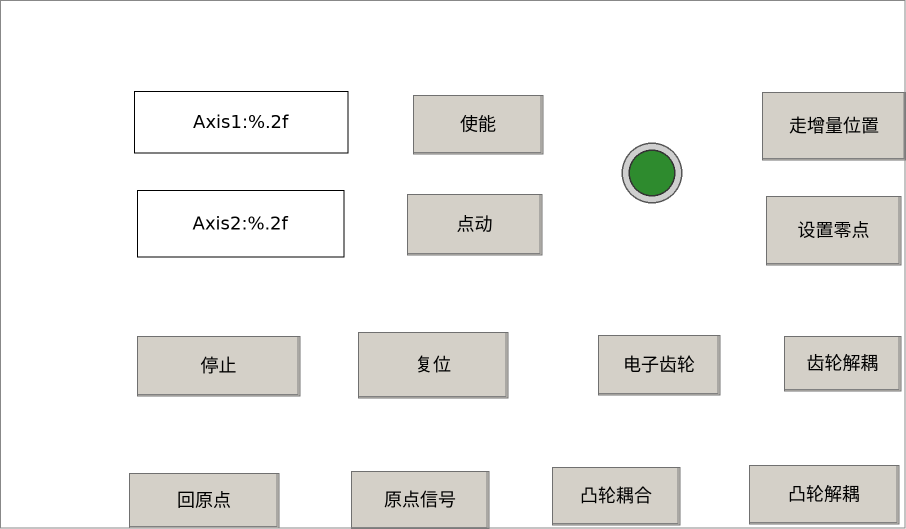
VISUALIZATION hmi  // 906x529
    Rectangle (134,91 214x62), "Axis1:%.2f", text variable: Motion01.Axis01.NcToPlc.ActPos
    Rectangle (137,190 207x67), "Axis2:%.2f", text variable: Motion01.Axis02.NcToPlc.ActPos
    Button (413,95 130x59), "使能"
        toggle Motion01.Power_Do
    Button (407,194 135x61), "点动"
        toggle Motion01.Jog_For
    Lamp1 (617,138 70x70), variable: Motion01.Axis01.NcToPlc.StateDWord.20, style: Lamp-Lamp1-Green
    Button (762,92 144x68), "走增量位置"
        tap Motion01.Move_Do
    Button (766,196 135x69), "设置零点"
        tap Motion01.Set_Do
    Button (137,336 163x60), "停止"
        tap Motion01.Stop_Do
    Button (358,332 150x66), "复位"
        tap Motion01.Reset_Do
    Button (598,335 122x60), "电子齿轮"
        tap Motion01.Gearin_Do
    Button (784,336 117x55), "齿轮解耦"
        tap Motion01.Gearout_Do
    Button (129,473 150x55), "回原点"
        tap Motion01.Home_Do
    Button (351,471 138x58), "原点信号"
        tap Motion01.Sensor
    Button (552,467 128x58), "凸轮耦合"
        tap Motion01.Cam_Do
    Button (749,465 150x59), "凸轮解耦"
        tap Motion01.Camout_Do
END_VISUALIZATION

(* stored: Version 1.1.0.1, ProductVersion 3.1.4024.10
   Visu hmi: Id {81cfe3a5-6fb4-4525-8e3f-daef0c871e81} *)
